PROGRAM SafetyCheck
VAR
	// slave robot information, including arm status and cartesian data
	m_slaveStatus AT %I* :ST_slaveStatus;
	
	// slave robot joint data
	m_slaveJointData AT %I* :ST_slaveJointData;
	
	// setup robot information
	m_setupStatus AT %I* :ST_SetupStatus;
	
	// setup robot joint data
	m_setupJointsData AT %I* :ST_SetupJointData;
	
	// master robot data, input from master controller box
	m_masterRobotData AT %I* : MSCommu_MasterStatus;
	
	// error check result
	m_safetyCheckData AT %Q* :ST_SafetyData;
	
	// Output cart status
	m_cartStatus AT%I* : ST_CartStatus;
	
	// cart joint data
	m_cartJointsData AT %I* :ST_CartJointData;
	
	//setup motor in_output to safety check
	m_setupMotorData AT %I* : ST_SetupMotorData;
	
	//slave motor in_output to safety check
	m_slaveMotorData AT %I* : ST_SlaveMotorData;
	
	//emergency stop and stop botton
	m_stopButton AT %I*: BOOL;
	m_emergencyStopButton AT %I*: BOOL;
	
	//warning tone
	m_warningTone AT %Q*:ARRAY [1..4] OF BOOL;
	
	//joystick Signal safety check
	m_joystickSignalIOSafetyCheck AT %I* : ARRAY [1..4] OF UDINT;
	
	//cart six-forceSensor
	m_sixForceSensor AT %I* : ARRAY [1..3] OF UDINT;
	
	//brake distance check outpurt
	m_brakeDistanceCheck AT %Q* : BOOL;
	
	i , j: INT;
	m_systemInitFlag:bool;
	m_SafetyCheck : Fb_SafetyCheck;
	m_clearFault : BOOL;
	m_checkVariable : ARRAY[1..g_maxNum] OF checkInputVariable;
	m_EtherCATCheck :ARRAY [1..g_maxNum,1..g_maxArmJoint] OF Fb_EtherCATCheck;
	m_EtherCATClearCRC :ARRAY [1..g_sArmNum] OF Fb_EtherCATCheck;
	m_RS232EtherCATState : ST_EtherCATState;
	
	//error robot data record
	m_dataRecord : Fb_dataRecord;
	
	// original position of remote center point when fisrt enter hold state
	m_dsrRcpPos :ARRAY[1..g_sArmNum] OF Vec3d;
	m_rcpPosErrCounts :ARRAY[1..g_sArmNum] OF INT := [4(0)];
	m_rcpPosErr :ARRAY[1..g_sArmNum] OF Vec3d;		// rcp position error
	m_motorEncoderSaltaValue : ARRAY [1..g_maxArmNum] OF vec13di;  
	
	m_armsRS:ARRAY [1..g_maxArmNum,1..50] OF RS;//复位优先双稳态器
	m_cartRS:ARRAY [1..50] OF RS;//复位优先双稳态器
	m_resetTon :ARRAY [1..g_maxArmNum,1..2] OF FB_TON;
	m_scopeArmNoReady : BOOL;
	m_joysticksTrigger : BOOL;
	// wait time before robot init  for ethercat to be statble 
	m_safetyCheckInitWaitTime : Vec5d;
	m_safetyCheckDriveOPWaitTime : LREAL:=0;
	m_safetyCheckReadFileWaitTime : LREAL:=0;
	
	m_EtherCATAllOP : BOOL:=FALSE;
	m_armEtherCATInOP : vec4b;
	m_moduleEtherCATInOPState : Vec5b;
	m_dumpEnergy : UDINT;
	
	m_mStopButton : FB_MasterStopButtonDetect;
	m_sStopButton : FB_MasterStopButtonDetect;
	
	//recipe read-write commands
	RecipeManCommands:   RecipeManCommands;
	m_bReadRecipeStep:   INT := 1;
	m_bWriteRecipeStep:   INT := 1;
	m_bReadRecipe:  BOOL := TRUE;
	m_bReadRecipeRecord:  BOOL := TRUE;
	
	m_bReadRecipeScope: BOOL := TRUE;
	
	m_bWriteRecipe: BOOL := FALSE;
	m_bWriteRecipeR: ARRAY [1..10] OF R_TRIG;
	m_ReturnDwordWrite : DWORD;
	m_loadConfigFileOK :BOOL :=FALSE;
	m_returnDwordRead:DWORD;
	m_returnDwordReadCart:DWORD;
	m_returnDwordReadMotorPara:DWORD;
	m_returnDwordReadReParam:DWORD;
	
	m_returnDwordReadScope:DWORD;
	
	m_caliFileWriteTon :ARRAY [1..g_sArmNum] OF TON ;
	m_linkPosWriteCaliData:ARRAY [1..4] OF ARRAY [1..8] OF TON ;
	m_powerBoxWriteCaliData:ARRAY [1..4] OF TON ;
	m_caliFileWriteTonOfCart :TON ;
	m_linkPosWriteCaliDataOfCart:ARRAY [1..8] OF TON ;

	
	//workHeart
	m_workHeartTon0 : TON;
	m_workHeartTon1 : TON;
	
	// flag if master are connected
	m_masterOnLine :BOOL :=FALSE;
	m_masterOnLineCheck :FB_masterConnectionCheck;
	
	//robot system operates sound 
	m_systemVoiceR:ARRAY [1..g_sArmNum,1..10] OF R_TRIG;
	m_systemVoiceF:ARRAY [1..g_sArmNum,1..10] OF F_TRIG;
	m_systemVoiceRS:ARRAY [1..g_sArmNum,1..10] OF RS;
	m_systemVoiceTon:ARRAY [1..g_sArmNum,1..10] OF FB_TON;
	m_checkArmKeepTriggerTon :ARRAY [1..g_sArmNum] OF FB_TON;
	m_trocarOnDetectTon:ARRAY [1..g_sArmNum] OF FB_TON;
	m_armStateLast:ARRAY[1..g_sArmNum] OF E_SlaveArmState;
	m_systemVoiceTriggerTime :TIME:=T#100MS;
	m_armKeepTriggerState :Vec4b;
	
	//read Net ID and Net port
	m_deviceNetIdReadOK : BOOL;
	m_bReadNetIdStep : INT := 1;
	m_bReadNetIdNum : INT := 1;
	m_bReadJntPortNum : INT := 1;
	m_getDeviceId :ARRAY [1..6] OF IOF_GetDeviceIDByName;
	m_getNetId :ARRAY [1..6] OF IOF_GetDeviceNetId;
	m_getBoxAddr:ARRAY [1..5,1..13] OF IOF_GetBoxAddrByName;
	m_readNetID: ARRAY[1..6] OF T_AmsNetId;
	m_readDeviceID : ARRAY [1..6]  OF UDINT;
	m_readJointNetPort:ARRAY[1..13] OF UINT;
END_VAR

// Faulty sound effect
m_warningTone := warningTone();
communicationCheck();
// reset data
m_deviceNetIdReadOK:=readDeviceNetId();
m_loadConfigFileOK:=loadConfigFile();
IF NOT(m_loadConfigFileOK) OR NOT m_deviceNetIdReadOK THEN
	m_safetyCheckReadFileWaitTime := m_safetyCheckReadFileWaitTime + g_safetyCheckCycleTime;
	IF m_safetyCheckReadFileWaitTime > g_robotSafetyReadFileWaitTime THEN
		GVL_interactUI.g_errIdType3:=checkFileAndNetId(m_loadConfigFileOK , m_deviceNetIdReadOK );
	END_IF
	RETURN;
END_IF
GVL_interactUI.g_systemVoice := systemVoice();

IF FALSE = m_systemInitFlag  THEN
	m_systemInitFlag := systemParaInit();
	RETURN;
END_IF

armSafetyCheckInputCast();

armSafetyCheckAllowed();

robotPromptMassageCast();

//robot record information
m_dataRecord.run(m_checkVariable , m_cartStatus , m_cartJointsData , m_setupStatus , m_slaveStatus , m_setupJointsData , m_slaveJointData );

//check EtherCAT status of arm and cart , if All EtherCAT is OP then start system safty check
IF FALSE = m_EtherCATAllOP THEN
	m_EtherCATAllOP := checkOPState();
END_IF

FOR i:=1  TO g_maxNum DO
	IF  NOT m_moduleEtherCATInOPState[i] AND NOT m_EtherCATAllOP THEN
		CONTINUE;
	END_IF
	
	// wait communication to be stable
	IF (m_safetyCheckInitWaitTime[i]<g_robotSafetyCheckWaitTime) THEN
		m_safetyCheckInitWaitTime[i] := m_safetyCheckInitWaitTime[i]+g_safetyCheckCycleTime;
	END_IF
	
	IF (m_safetyCheckInitWaitTime[i]>=g_robotSafetyCheckWaitTime) THEN
		m_SafetyCheck.systemSafetyCheck(i,m_checkVariable,m_cartJointsData,m_setupJointsData,m_slaveJointData);
	END_IF
END_FOR

//error flag to control
readErrFlag();

//Fault code for UI
m_SafetyCheck.errCodeUpdating();

//The fault code is sent to the UI
GVL_interactUI.g_errIdType3:=m_SafetyCheck.o_ErrCode[3];
GVL_interactUI.g_errIdType2:=m_SafetyCheck.o_ErrCode[2];
GVL_interactUI.g_errIdType1:=m_SafetyCheck.o_ErrCode[1];
GVL_interactUI.g_errIdType0:=m_SafetyCheck.o_ErrCode[0];
GVL_interactUI.g_popupErrorArm1 := m_SafetyCheck.m_armErrCodePopup[1];
GVL_interactUI.g_popupErrorArm2 := m_SafetyCheck.m_armErrCodePopup[2];
GVL_interactUI.g_popupErrorArm3 := m_SafetyCheck.m_armErrCodePopup[3];
GVL_interactUI.g_popupErrorArm4 := m_SafetyCheck.m_armErrCodePopup[4];

//clear fault
clearErrorFault();

METHOD armSafetyCheckAllowed : BOOL
VAR_INPUT
END_VAR
VAR
	i , j : INT; 
END_VAR
FOR i := 1 TO g_maxArmNum DO
	FOR j := 1 TO g_maxArmJoint DO
		IF j > 5 THEN
			//fault code 16#3003 
			m_SafetyCheck.checkPermit[i].m_linkEncErr[j] := m_checkVariable[i].m_slaveDriverInput[j-g_setupJntNum].m_statusWord<>0;
			//fault code 16#2002
			m_SafetyCheck.checkPermit[i].m_armJntFollowErr[j] := m_checkVariable[i].m_slaveDriverInput[j-g_setupJntNum].m_statusWord = DriverStatusWord_OP ;
			//fault code 16#200B
			m_SafetyCheck.checkPermit[i].m_jntCurrentCtrlErr[j] :=SlaveArmControl.m_slaveRobot.m_armCtrlCmds[i].m_jntEnableFlag[j-g_setupJntNum]  = DriverOPMode_Trq AND m_slaveMotorData.m_slaveMotorOutput[i,j-g_setupJntNum].m_opMode = DriverOPMode_Trq ;
		ELSE
			//fault code 16#3003 
			m_SafetyCheck.checkPermit[i].m_linkEncErr[j] := m_checkVariable[i].m_setupDriverInput[j].m_statusWord<>0;
			//fault code 16#2002
			m_SafetyCheck.checkPermit[i].m_armJntFollowErr[j] := m_checkVariable[i].m_setupDriverInput[j].m_statusWord = DriverStatusWord_OP AND j > 2;
			//fault code 16#200B
			m_SafetyCheck.checkPermit[i].m_jntCurrentCtrlErr[j] := SetupArmControl.m_setupRobot.m_armCtrlCmds[i].m_jntEnableFlag[j] = DriverOPMode_Trq AND m_setupMotorData.m_setupMotorOutput[i,j].m_opMode = DriverOPMode_Trq AND j > 2;
			
		END_IF
		//fault code 16#3002
		m_SafetyCheck.checkPermit[i].m_jntStatusErr[j] := TRUE;
		//fault code 16#3004
		m_SafetyCheck.checkPermit[i].m_driveErr[j] := TRUE;
		//fault code 16#3005
		m_SafetyCheck.checkPermit[i].m_armJntEncErr[j] := m_checkVariable[i].m_setupDriverInput[j].m_statusWord<>0;
		//fault code 16#3006
		m_SafetyCheck.checkPermit[i].m_outOfLimit[j] := m_checkVariable[i].m_setupDriverInput[j].m_statusWord<>0;
		//fault code 16#3008
		m_SafetyCheck.checkPermit[i].m_motPhieErr[j] := TRUE;
		//fault code 16#3009
		m_SafetyCheck.checkPermit[i].m_springBreakageCheck := TRUE;//m_checkVariable[i].m_setupDriverInput[j].m_statusWord<>0 ;
		//fault code 16#2003
		m_SafetyCheck.checkPermit[i].m_jntVelErr[j] := TRUE;
		//fault code 16#2004
		m_SafetyCheck.checkPermit[i].m_spacePoseErr := m_slaveStatus.m_armState[i] = SlaveArmState_MasterSlave;
		//fault code 16#2005
		m_SafetyCheck.checkPermit[i].m_jntCurrentErr[j] := TRUE;
		//fault code 16#2007
		m_SafetyCheck.checkPermit[i].m_fixedPointErr :=m_slaveStatus.m_armState[i] = SlaveArmState_MasterSlave;
		//fault code 16#2008
		m_SafetyCheck.checkPermit[i].m_cmdJntSaltation[j] := m_slaveStatus.m_armState[i] = SlaveArmState_MasterSlave;
		//fault code 16#200A
		m_SafetyCheck.checkPermit[i].m_simCmdSalta := m_slaveStatus.m_armState[i] = SlaveArmState_MasterSlave;
		//fault code 16#200F
		m_SafetyCheck.checkPermit[i].m_instruOpenAngle := FALSE;
		//fault code 16#2013
		m_SafetyCheck.checkPermit[i].m_jntLimitErr := m_slaveStatus.m_armState[i] = SlaveArmState_MasterSlave;
	END_FOR
END_FOR
END_METHOD

METHOD armSafetyCheckInputCast : BOOL
VAR_INPUT
END_VAR

VAR
	i , j: INT; 
END_VAR
FOR i := 1 TO g_maxArmNum DO
	//emergency stop 、stop button and ui stop 
	m_checkVariable[i].EmergencyStop := m_emergencyStopButton;
	m_checkVariable[i].PCStopButton := GVL_interactUI.g_stopButtonFormUI;
	m_checkVariable[i].SlaveStopButton := m_sStopButton.run(m_stopButton);
	m_checkVariable[i].MasterStopButton := m_mStopButton.run(m_masterRobotData.m_masterStopButton);
	
	IF NOT(m_slaveStatus.m_armState[i] = SlaveArmState_MasterSlave OR m_slaveStatus.m_armState[i] = SlaveArmState_EndoScope) THEN
		m_dsrRcpPos[i] := m_setupStatus.m_rcPos[i];
	END_IF
	m_checkVariable[i].m_rcpCheck := m_SafetyCheck.rcpErrCheck(m_dsrRcpPos[i],  m_setupStatus.m_rcPos[i], m_rcpPosErrCounts[i] ,m_rcpPosErr[i]);
	m_checkVariable[i].m_spacePoseErr := m_SafetyCheck.rotErrCheck(m_slaveStatus.m_masterSlavePoseError[i]);
	m_checkVariable[i].m_cmdArmPos := m_slaveStatus.m_simDHJntPos[i];

	//slave robot input cast
	FOR j:=1 TO  g_sJntNum DO 		
		m_checkVariable[i].m_slaveDriverInput[j] := m_slaveMotorData.m_slaveMotorInput[i,j];
		m_checkVariable[i].m_slaveDriverOutput[j] := m_slaveMotorData.m_slaveMotorOutput[i,j];
		m_checkVariable[i].m_EtherCATState[j+g_setupJntNum] := m_EtherCATCheck[i,j+g_setupJntNum].EtherCATVerify(GVL_SystemParameters.g_slaveArmNetID[i],GVL_SystemParameters.g_slaveJointNetPort[i,j]);
		m_checkVariable[i].m_motorEncoderSaltaValue[j+g_setupJntNum] := m_slaveMotorData.m_motorEncSalta[i][j];
	END_FOR
	
	//setup robot input cast
	FOR j:=1 TO  g_setupJntNum DO 	
		m_checkVariable[i].m_setupDriverInput[j] := m_setupMotorData.m_setupMotorInput[i,j];
		m_checkVariable[i].m_setupDriverOutput[j] := m_setupMotorData.m_setupMotorOutput[i,j];
		m_checkVariable[i].m_EtherCATState[j] := m_EtherCATCheck[i,j].EtherCATVerify(GVL_SystemParameters.g_slaveArmNetID[i],GVL_SystemParameters.g_setupJointNetPort[i,j]);
		m_checkVariable[i].m_motorEncoderSaltaValue[j] := m_setupMotorData.m_motorEncSalta[i][j];
	END_FOR
END_FOR


//setup robot in-out variable cast
FOR j:=1 TO  g_cartJntNum DO
	m_checkVariable[5].EmergencyStop := m_emergencyStopButton;
	m_checkVariable[5].PCStopButton := GVL_interactUI.g_stopButtonFormUI;
	m_checkVariable[5].SlaveStopButton := m_sStopButton.run(m_stopButton);
	m_checkVariable[5].m_cartDriverInput[j] := CartControl.m_cartRobot.m_slaveCart.m_cartJoints[j].m_motorInputs;
	m_checkVariable[5].m_cartDriverOutput[j] := CartControl.m_cartRobot.m_slaveCart.m_cartJoints[j].m_motorOutputs;
	m_checkVariable[5].m_cartEtherCATState[j] := m_EtherCATCheck[5,j].EtherCATVerify(GVL_SystemParameters.g_slaveCartNetID,GVL_SystemParameters.g_cartJointNetPort[j]);
END_FOR

//RS232 communication state
m_RS232EtherCATState := m_EtherCATCheck[5,9].EtherCATVerify(GVL_SystemParameters.g_slaveCartNetID,GVL_SystemParameters.g_cartJointNetPort[5]+1);

//output to ui
Gvl_io.g_emergencyStopButton := m_emergencyStopButton;
Gvl_io.g_stopButton := m_stopButton;
END_METHOD

METHOD checkEtherCATAll : BOOL
VAR_IN_OUT CONSTANT
	i_EtherCATState: ARRAY [1..g_maxNum] OF checkInputVariable;
END_VAR
VAR_OUTPUT
	o_EtherCATInOP : BOOL;
	o_armEtherCATInOP : vec4b;
	o_cartEtherCATAllOP : BOOL;
END_VAR

VAR
	i , j :INT;
END_VAR
FOR i := 1 TO g_sArmNum DO
	FOR j := 1 TO g_maxArmJoint DO
		//m_EtherCATCheck[i,j].setSlaveStatus(GVL_SlaveJointEncoderCaliData.g_slaveArmNetID[i],g_JointNetPort[j]);
	END_FOR
END_FOR

o_EtherCATInOP := TRUE;
FOR i := 1 TO g_sArmNum DO
	o_armEtherCATInOP[i] := TRUE;
	FOR j := 1 TO g_maxArmJoint DO
		IF FALSE = i_EtherCATState[i].m_EtherCATState[j].EtherCATState AND i <> GVL_interactUI.g_armIsDisable THEN
			o_armEtherCATInOP[i] := FALSE;
			o_EtherCATInOP := FALSE;
			EXIT;
		END_IF
	END_FOR
	IF NOT o_armEtherCATInOP[i] OR NOT o_EtherCATInOP THEN
		EXIT;
	END_IF
END_FOR

FOR j := 1 TO g_maxCartJoint DO
	//m_EtherCATCheck[5,j].setSlaveStatus(GVL_CartJointEncoderCaliData.g_slaveCartNetID,GVL_CartJointEncoderCaliData.g_slaveCartJointNetPort[j]);
END_FOR

o_cartEtherCATAllOP := TRUE;
FOR j := 1 TO g_maxCartJoint DO
	IF FALSE = i_EtherCATState[5].m_cartEtherCATState[j].EtherCATState THEN
		o_cartEtherCATAllOP := FALSE;
		EXIT;
	END_IF
END_FOR
END_METHOD

METHOD checkFileAndNetId : UDINT
VAR_IN_OUT CONSTANT
	i_readConfigFileStatus :BOOL;
	i_readDeviceNetIdStatus :BOOL;
END_VAR

IF NOT i_readConfigFileStatus OR NOT i_readDeviceNetIdStatus THEN
	checkFileAndNetId:=SHL(16#0C,24)+SHL(0,16)+16#300A;
END_IF
END_METHOD

METHOD checkOPState : BOOL
VAR_INPUT
END_VAR
IF (NOT m_safetyCheckData.m_armEtherCATAllOP OR NOT m_safetyCheckData.m_cartEtherCATAllOP) THEN
	m_safetyCheckDriveOPWaitTime := m_safetyCheckDriveOPWaitTime+g_safetyCheckCycleTime;
	IF m_safetyCheckDriveOPWaitTime > g_robotSafetyDriveOPWaitTime THEN
		 m_SafetyCheck.checkOPStatus(m_moduleEtherCATInOPState);
	END_IF
	RETURN;
END_IF
checkOPState := TRUE;
m_SafetyCheck.resetOPErrCode();
END_METHOD

METHOD clearErrorFault : BOOL
VAR_INPUT
END_VAR
VAR_STAT
	clearFaultTime : FB_TON;
END_VAR
// clear CRC lost frame
m_clearFault := GVL_interactUI.g_uiFaultReset=1 OR m_masterRobotData.m_uiResetFault = 1;
clearFaultTime(IN:= m_clearFault, PT:= T#2MS, Q=> , ET=> );
FOR i:=1 TO g_sArmNum DO 
	m_EtherCATClearCRC[i].clearCRCError(GVL_SystemParameters.g_slaveArmNetID[i],clearFault);
END_FOR
//clear fault
IF m_clearFault THEN
	m_SafetyCheck.errFlagReset();
	IF clearFaultTime.Q THEN
		GVL_interactUI.g_uiFaultReset := 0;
	END_IF
END_IF
END_METHOD

PROPERTY clearFault : BOOL;
GET
clearFault := m_clearFault;
END_GET
END_PROPERTY

METHOD communicationCheck : BOOL
VAR_INPUT
END_VAR
VAR
	i : INT;
END_VAR
checkEtherCATAll(m_checkVariable , o_EtherCATInOP=>m_safetyCheckData.m_armEtherCATAllOP,o_armEtherCATInOP=> m_armEtherCATInOP, o_cartEtherCATAllOP=> m_safetyCheckData.m_cartEtherCATAllOP );
FOR i := 1 TO g_sArmNum DO
	m_moduleEtherCATInOPState[i] := m_armEtherCATInOP[i];
END_FOR
m_moduleEtherCATInOPState[5] := m_safetyCheckData.m_cartEtherCATAllOP;

m_brakeDistanceCheck :=NOT UINT_TO_BOOL( GVL_interactUI.g_stopButtonFormUI);

//work heart
m_workHeartTon0(IN:= GVL_interactUI.g_heartBeat = 1, PT:= T#1S, Q=> , ET=> );
m_workHeartTon1(IN:= GVL_interactUI.g_heartBeat = 0, PT:= T#1S, Q=> , ET=> );
IF m_workHeartTon0.Q THEN
	GVL_interactUI.g_heartBeat :=0 ;
ELSIF m_workHeartTon1.Q THEN
	GVL_interactUI.g_heartBeat  :=1 ;
END_IF

//master online
m_masterOnLine := m_masterOnLineCheck.check(m_masterRobotData.m_heartBeat );

GVL_interactUI.g_slaveRunAlone := NOT m_masterOnLine;
END_METHOD

METHOD jointEncoderCaliCast : BOOL
VAR_INPUT
	armIdx : INT;
END_VAR
VAR 
	i : INT;
END_VAR

FOR i := 1 TO 8 DO
	m_linkPosWriteCaliData[armIdx][i](IN:= GVL_armCali.g_linkPosWriteCaliData[armIdx][i], PT:= T#3S, Q=> GVL_armCali.g_linkPosWriteCaliDataTrigger[armIdx][i], ET=> );
	IF GVL_armCali.g_linkPosWriteCaliDataTrigger[armIdx][i] THEN
		IF i<=5 THEN
			GVL_SetupJointEncoderCaliData.g_minLinkEncoder[armIdx,i] := GVL_armCali.g_linkLimitFristPos[armIdx][i];
			GVL_SetupJointEncoderCaliData.g_maxLinkEncoder[armIdx,i] := GVL_armCali.g_linkLimitSecondPos[armIdx][i];
			GVL_SetupJointEncoderCaliData.g_caliLinkEncoder[armIdx,i] := GVL_armCali.g_linkHomePos[armIdx][i];
			GVL_SetupJointEncoderCaliData.g_linkEncZeroCross[armIdx,i] := GVL_armCali.g_linkZeroCrossOrNot[armIdx][i];
		ELSE
			GVL_SlaveJointEncoderCaliData.g_minLinkEncoder[armIdx,i-5] := GVL_armCali.g_linkLimitFristPos[armIdx][i];
			GVL_SlaveJointEncoderCaliData.g_maxLinkEncoder[armIdx,i-5] := GVL_armCali.g_linkLimitSecondPos[armIdx][i];
			GVL_SlaveJointEncoderCaliData.g_caliLinkEncoder[armIdx,i-5] := GVL_armCali.g_linkHomePos[armIdx][i];
			GVL_SlaveJointEncoderCaliData.g_linkEncZeroCross[armIdx,i-5] := GVL_armCali.g_linkZeroCrossOrNot[armIdx][i];
		END_IF
	END_IF
END_FOR
FOR i := 1 TO 5 DO
	m_powerBoxWriteCaliData[armIdx](IN:= GVL_armCali.g_powerBoxPosWrite[armIdx], PT:= T#3S, Q=>GVL_armCali.g_powerBoxPosWriteTrigger[armIdx] , ET=> );
	IF GVL_armCali.g_powerBoxPosWriteTrigger[armIdx] THEN
		GVL_SlaveJointEncoderCaliData.g_caliLinkEncoder[armIdx,i+3] := GVL_armCali.g_powerBoxLinkHomePos[armIdx][i];
	END_IF
END_FOR

FOR i := 1 TO g_cartJntNum DO
	m_linkPosWriteCaliDataOfCart[i](IN:= GVL_armCali.g_linkPosWriteCaliDataOfCart[i], PT:= T#3S, Q=> GVL_armCali.g_linkPosWriteCaliDataTriggerOfCart[i], ET=> );
	IF GVL_armCali.g_linkPosWriteCaliDataTriggerOfCart[i] THEN
		GVL_CartJointEncoderCaliData.g_minLinkEncoder[i] := GVL_armCali.g_linkLimitFristPosOfCart[i];
		GVL_CartJointEncoderCaliData.g_maxLinkEncoder[i] := GVL_armCali.g_linkLimitSecondPosOfCart[i];
		GVL_CartJointEncoderCaliData.g_caliLinkEncoder[i] := GVL_armCali.g_linkHomePosOfCart[i];
		GVL_CartJointEncoderCaliData.g_linkEncZeroCross[i] := GVL_armCali.g_linkZeroCrossOrNotOfCart[i];
	END_IF
END_FOR
END_METHOD

METHOD joystickAdjust : BOOL
VAR_IN_OUT CONSTANT
	i_joystickValue : ARRAY [1..4] OF UDINT;
END_VAR

VAR
	i : INT;
END_VAR

FOR i := 1 TO 4 DO
	IF  (i_joystickValue[i]>1 AND i_joystickValue[i]<(512-50)) OR i_joystickValue[i] > (512+50) THEN
		joystickAdjust := TRUE;
		EXIT;
	END_IF
END_FOR
END_METHOD

METHOD loadConfigFile : BOOL
VAR
	i:INT;
	recordParam : BOOL;
	ReturnDwordWrite :DWORD;
END_VAR
//read recipe
IF (m_bReadRecipeStep<=12 AND m_bReadRecipeStep>0) THEN
	//The method loads a recipe from the specified recipe file.  It subsequently writes the recipe into the PLC variables.
    m_returnDwordRead:=RecipeManCommands.LoadAndWriteRecipe(RecipeDefinitionName:=GVL_SystemParameters.RecipeDefinitionName[m_bReadRecipeStep] , RecipeName:='RecipeRecord');
	IF m_returnDwordRead = ERR_OK THEN
		m_bReadRecipeStep:=m_bReadRecipeStep+1; 
	END_IF
END_IF 
loadConfigFile := m_bReadRecipeStep>12;


// read Recipe 
IF (m_bReadRecipe) THEN
	//The method loads a recipe from the specified recipe file.  It subsequently writes the recipe into the PLC variables.
     m_returnDwordReadCart:=RecipeManCommands.LoadAndWriteRecipe(RecipeDefinitionName:=GVL_SystemParameters.RecipeDefinitionNameCart, RecipeName:='RecipeRecord');	 
     m_returnDwordReadMotorPara:=RecipeManCommands.LoadAndWriteRecipe(RecipeDefinitionName:=GVL_SystemParameters.RecipeDefinitionNameMotorPara, RecipeName:='RecipeRecord');	
	m_bReadRecipe:=FALSE; 
END_IF
loadConfigFile := loadConfigFile AND (m_returnDwordReadCart = ERR_OK) AND m_returnDwordReadMotorPara = ERR_OK;

//read endoscope parameters
IF m_bReadRecipeScope THEN
	m_returnDwordReadScope:=RecipeManCommands.LoadAndWriteRecipe(RecipeDefinitionName:=GVL_SystemParameters.RecipeDefinitionNameScope, RecipeName:='RecipeRecord');	 
	m_bReadRecipeScope := FALSE;
END_IF
loadConfigFile := loadConfigFile AND m_returnDwordReadScope = ERR_OK;

//read robot record parameters
IF m_bReadRecipeRecord THEN
	m_returnDwordReadReParam:=RecipeManCommands.LoadAndWriteRecipe(RecipeDefinitionName:=GVL_SystemParameters.RecipeDefinitionNameRecordParam, RecipeName:='RecipeRecord');	 
	m_bReadRecipeRecord := FALSE;
END_IF


//write recipe
FOR i := 1 TO g_sArmNum DO
	jointEncoderCaliCast(i);
	m_caliFileWriteTon[i](IN:=GVL_armCali.g_caliDataWrite[i], PT:= T#3S, Q=> GVL_armCali.g_caliDataWriteTrigger[i], ET=> );
	IF GVL_armCali.g_caliDataWriteTrigger[i] THEN
		//This method creates a new recipe in the specified recipe definition. It subsequently reads the current PLC values into the new recipe and saves it as a recipe file with a standard name.
	 	RecipeManCommands.CreateRecipe(RecipeDefinitionName:=GVL_SystemParameters.RecipeDefinitionName[i] , RecipeName:='RecipeRecord' );
	 	ReturnDwordWrite:=RecipeManCommands.ReadAndSaveRecipe(RecipeDefinitionName:=GVL_SystemParameters.RecipeDefinitionName[i] , RecipeName:='RecipeRecord' );
	END_IF
END_FOR

m_caliFileWriteTonOfCart(IN:= GVL_armCali.g_caliDataWriteOfCart, PT:= T#3S, Q=> GVL_armCali.g_caliDataWriteTriggerOfCart, ET=> );
IF GVL_armCali.g_caliDataWriteTriggerOfCart THEN
	//This method creates a new recipe in the specified recipe definition. It subsequently reads the current PLC values into the new recipe and saves it as a recipe file with a standard name.
	 RecipeManCommands.CreateRecipe(RecipeDefinitionName:=GVL_SystemParameters.RecipeDefinitionNameCart , RecipeName:='RecipeRecord' );
	 ReturnDwordWrite:=RecipeManCommands.ReadAndSaveRecipe(RecipeDefinitionName:=GVL_SystemParameters.RecipeDefinitionNameCart , RecipeName:='RecipeRecord' );
	 m_bWriteRecipe:=FALSE;
END_IF

//write robot record parameters
FOR i := 1 TO g_sArmNum DO
	m_bWriteRecipeR[i](CLK:= MEMCMP(ADR(m_setupMotorData.m_jnt3MoveDistanceRecord[i]),ADR(m_setupMotorData.m_jnt3MoveDistance[i]),SIZEOF(m_setupMotorData.m_jnt3MoveDistanceRecord[i])) = 0, Q=> );
END_FOR
m_bWriteRecipeR[5](CLK:= MEMCMP(ADR(m_cartStatus.m_cartDriveForceOffset),ADR(m_cartStatus.m_cartDriveForceRecord),SIZEOF(m_cartStatus.m_cartDriveForceRecord)) = 0, Q=> );

m_bWriteRecipe := FALSE;
FOR i := 1 TO 10 DO
	IF m_bWriteRecipeR[i].Q THEN
		m_bWriteRecipe := m_bWriteRecipeR[i].Q;
		EXIT;
	END_IF
END_FOR

IF m_bWriteRecipe THEN
	 RecipeManCommands.CreateRecipe(RecipeDefinitionName:=GVL_SystemParameters.RecipeDefinitionNameRecordParam , RecipeName:='RecipeRecord' );
	 m_ReturnDwordWrite:=RecipeManCommands.ReadAndSaveRecipe(RecipeDefinitionName:=GVL_SystemParameters.RecipeDefinitionNameRecordParam , RecipeName:='RecipeRecord' );
END_IF
END_METHOD

METHOD readDeviceNetId : BOOL
VAR_INPUT
END_VAR
//read device NetId
CASE m_bReadNetIdStep OF
	1 ://read the device ID using the device name
		m_getDeviceId[m_bReadNetIdNum](NETID:= , DEVICENAME:= GVL_SystemParameters.g_deviceName[m_bReadNetIdNum], START:= TRUE, TMOUT:= , BUSY=> , ERR=> , ERRID=> , DEVICEID=> m_readDeviceID[m_bReadNetIdNum]);
		IF m_readDeviceID[m_bReadNetIdNum] <> 0 THEN
			m_bReadNetIdNum := m_bReadNetIdNum + 1;
			IF m_bReadNetIdNum > 6 THEN
				m_bReadNetIdNum:=1;
				m_bReadNetIdStep := 2;
			END_IF
		END_IF
		
	2:
		m_getNetId[m_bReadNetIdNum](NETID:= , DEVICEID:= m_readDeviceID[m_bReadNetIdNum], START:= TRUE, TMOUT:= , BUSY=> , ERR=> , ERRID=> , DeviceNetId=> m_readNetID[m_bReadNetIdNum]);
		IF m_readNetID[m_bReadNetIdNum] <> '' THEN
			IF m_bReadNetIdNum <= 4 THEN
				GVL_SystemParameters.g_slaveArmNetID [m_bReadNetIdNum] := m_readNetID[m_bReadNetIdNum];
				IF GVL_SystemParameters.g_slaveArmNetID [m_bReadNetIdNum] <> '' THEN
					m_bReadNetIdNum := m_bReadNetIdNum + 1;
				END_IF
			ELSIF m_bReadNetIdNum = 5 THEN
				GVL_SystemParameters.g_slaveCartNetID := m_readNetID[m_bReadNetIdNum];	
				IF GVL_SystemParameters.g_slaveCartNetID<> '' THEN
					m_bReadNetIdNum := m_bReadNetIdNum + 1;
				END_IF
			ELSIF m_bReadNetIdNum = 6 THEN
				GVL_SystemParameters.g_slaveMSComNetID := m_readNetID[m_bReadNetIdNum];	
				IF GVL_SystemParameters.g_slaveMSComNetID<> '' THEN
					m_bReadNetIdNum := m_bReadNetIdNum + 1;
				END_IF
			END_IF
			
			IF m_bReadNetIdNum > 6 THEN
				m_bReadNetIdNum:=1;
				m_bReadJntPortNum := 1;
				m_bReadNetIdStep := 3;
			END_IF
		END_IF
		
	3:
		IF m_bReadNetIdNum <= 4 THEN
			m_getBoxAddr[m_bReadNetIdNum,m_bReadJntPortNum](NETID:= , DEVICEID:= m_readDeviceID[m_bReadNetIdNum], BOXNAME:=GVL_SystemParameters.g_armDeviceJntName[m_bReadJntPortNum] , START:= TRUE, TMOUT:= , BUSY=> , ERR=> , ERRID=> , BOXADDR=> m_readJointNetPort[m_bReadJntPortNum]);
			IF m_bReadJntPortNum <= 5 THEN
				GVL_SystemParameters.g_setupJointNetPort[m_bReadNetIdNum,m_bReadJntPortNum] := m_readJointNetPort[m_bReadJntPortNum];
				IF GVL_SystemParameters.g_setupJointNetPort[m_bReadNetIdNum,m_bReadJntPortNum] <> 0 THEN
					m_bReadJntPortNum := m_bReadJntPortNum +1;
				END_IF
			ELSE
				GVL_SystemParameters.g_slaveJointNetPort[m_bReadNetIdNum,m_bReadJntPortNum-5]:= m_readJointNetPort[m_bReadJntPortNum];
				IF GVL_SystemParameters.g_slaveJointNetPort[m_bReadNetIdNum,m_bReadJntPortNum-5] <> 0 THEN
					m_bReadJntPortNum := m_bReadJntPortNum +1;
				END_IF
			END_IF
			IF m_bReadJntPortNum > 13 THEN
				m_bReadJntPortNum := 1;
				m_bReadNetIdNum := m_bReadNetIdNum + 1;
			END_IF
		ELSIF m_bReadNetIdNum = 5 THEN
			m_getBoxAddr[m_bReadNetIdNum,m_bReadJntPortNum](NETID:= , DEVICEID:= m_readDeviceID[m_bReadNetIdNum], BOXNAME:=GVL_SystemParameters.g_cartDeviceJntName[m_bReadJntPortNum] , START:= TRUE, TMOUT:= , BUSY=> , ERR=> , ERRID=> , BOXADDR=> m_readJointNetPort[m_bReadJntPortNum]);
				GVL_SystemParameters.g_cartJointNetPort[m_bReadJntPortNum] := m_readJointNetPort[m_bReadJntPortNum];
				IF GVL_SystemParameters.g_cartJointNetPort[m_bReadJntPortNum] <> 0 THEN
					m_bReadJntPortNum := m_bReadJntPortNum +1;
				END_IF
				IF m_bReadJntPortNum > 8 THEN
					m_bReadJntPortNum := 1;
					m_bReadNetIdNum := m_bReadNetIdNum + 1;
				END_IF
		END_IF
       
		IF m_bReadNetIdNum > 5 THEN
			m_bReadNetIdNum:=1;
			m_bReadNetIdStep := -1;
		END_IF
	
	-1:
		readDeviceNetId := TRUE;
END_CASE
END_METHOD

METHOD readErrFlag : BOOL
VAR_INPUT
END_VAR
FOR i:=1  TO g_sArmNum DO
	m_safetyCheckData.m_slaveErrFlag[i] := m_SafetyCheck.m_armErrFlag[i,2] OR m_SafetyCheck.m_armErrFlag[i,3];
	m_safetyCheckData.m_setupErrFlag[i] := m_SafetyCheck.m_armErrFlag[i,2] OR m_SafetyCheck.m_armErrFlag[i,3];
END_FOR


GVL_interactUI.g_slaveRecoverErrFlag := BOOL_TO_INT(((m_SafetyCheck.m_armErrFlag[1,2] AND GVL_interactUI.g_armIsDisable<>1) OR (m_SafetyCheck.m_armErrFlag[2,2] AND GVL_interactUI.g_armIsDisable<>2)
												 OR (m_SafetyCheck.m_armErrFlag[3,2] AND GVL_interactUI.g_armIsDisable<>3) OR (m_SafetyCheck.m_armErrFlag[4,2] AND GVL_interactUI.g_armIsDisable<>4)
														OR m_SafetyCheck.m_armErrFlag[g_cartNum,2] OR m_SafetyCheck.m_jntErrFlag[g_cartNum,0,2]) AND GVL_interactUI.g_slaveRunAlone) ;

//cart error flag
m_safetyCheckData.m_cartErrFlag := m_SafetyCheck.m_armErrFlag[g_cartNum,2] OR m_SafetyCheck.m_armErrFlag[g_cartNum,3];
//cart stead foot error flag
m_safetyCheckData.m_cartSteadyFootErr := m_SafetyCheck.m_jntErrFlag[g_cartNum,1,2] OR m_SafetyCheck.m_jntErrFlag[g_cartNum,1,3] 
																	OR m_SafetyCheck.m_jntErrFlag[g_cartNum,2,2] OR m_SafetyCheck.m_jntErrFlag[g_cartNum,2,3] OR m_SafetyCheck.m_jntErrFlag[g_cartNum,0,3];
//cart wheel error flag
m_safetyCheckData.m_cartWheelErr := m_SafetyCheck.m_jntErrFlag[g_cartNum,3,2] OR m_SafetyCheck.m_jntErrFlag[g_cartNum,3,3]
																OR m_SafetyCheck.m_jntErrFlag[g_cartNum,4,2] OR m_SafetyCheck.m_jntErrFlag[g_cartNum,4,3] OR m_SafetyCheck.m_stopButtonTrigger OR m_SafetyCheck.m_jntErrFlag[g_cartNum,0,3];
//cart stand column error flag
m_safetyCheckData.m_cartStandColumnErr := m_SafetyCheck.m_jntErrFlag[g_cartNum,5,2] OR m_SafetyCheck.m_jntErrFlag[g_cartNum,5,3] OR m_SafetyCheck.m_stopButtonTrigger OR m_SafetyCheck.m_jntErrFlag[g_cartNum,0,3];
//cart adjust joint contains 6, 7, and 8 joints
m_safetyCheckData.m_cartAdjustErr := m_SafetyCheck.m_jntErrFlag[g_cartNum,6,2] OR m_SafetyCheck.m_jntErrFlag[g_cartNum,6,3] 
															OR m_SafetyCheck.m_jntErrFlag[g_cartNum,7,2] OR m_SafetyCheck.m_jntErrFlag[g_cartNum,7,3]
															OR m_SafetyCheck.m_jntErrFlag[g_cartNum,8,2] OR m_SafetyCheck.m_jntErrFlag[g_cartNum,8,3] OR m_SafetyCheck.m_stopButtonTrigger OR m_SafetyCheck.m_jntErrFlag[g_cartNum,0,3];
//cart overhang error flag
m_safetyCheckData.m_cartOverhangErr := m_SafetyCheck.m_jntErrFlag[g_cartNum,8,2] OR m_SafetyCheck.m_jntErrFlag[g_cartNum,8,3] OR m_SafetyCheck.m_stopButtonTrigger OR m_SafetyCheck.m_jntErrFlag[g_cartNum,0,3];
END_METHOD

METHOD robotPromptMassageCast : BOOL
VAR_IN_OUT CONSTANT
END_VAR

VAR
	i : UDINT;
	m_uiCtrlAdjustFlag : BOOL;
	m_uiCtrlJoystickEnable : BOOL;
	instrument: INT;
	robotSelfCheckPass : BOOL;
	teleSlaveArmIdx : ARRAY [1..2] OF INT;
	panelMountedFlag : Vec4b;
	scopeNoReady : BOOL;
END_VAR
FOR i := 1 TO 4 DO
	//0*1021
	m_armsRS[i,1](SET:= m_slaveStatus.m_panelClampErrId[i]=1, 
							RESET1:= NOT m_slaveStatus.m_panelInstallStatus[i], 
							Q1=> m_checkVariable[i].m_promptStatus[1]);
	m_checkVariable[i].m_promptLocation[1] := i + 3;
							
	//0*1022		
	m_armsRS[i,2](SET:= m_slaveStatus.m_panelClampErrId[i]=2, 
							RESET1:= NOT m_slaveStatus.m_panelInstallStatus[i], 
							Q1=> m_checkVariable[i].m_promptStatus[2]);
	m_checkVariable[i].m_promptLocation[2] := i + 3;
	
	//0*1023				
	m_armsRS[i,3](SET:= m_slaveStatus.m_instruReadErrId[i]=1 AND m_slaveStatus.m_selfCheckPass[i], 
							RESET1:= NOT m_armsRS[i,3].SET OR NOT m_slaveStatus.m_instruInstallStatus[i] , 
							Q1=> m_checkVariable[i].m_promptStatus[3]);
	m_checkVariable[i].m_promptLocation[3] := i + 3;
						
	//0*1024	
	m_armsRS[i,4](SET:= m_slaveStatus.m_instruReadErrId[i]=2 AND m_slaveStatus.m_selfCheckPass[i],
							RESET1:=NOT m_armsRS[i,4].SET OR NOT m_slaveStatus.m_instruInstallStatus[i], 
							Q1=> m_checkVariable[i].m_promptStatus[4]);
	m_checkVariable[i].m_promptLocation[4] := i + 3;
	
	//0*1025
	m_armsRS[i,5](SET:= m_slaveStatus.m_instruClampErrId[i]=1 AND m_slaveStatus.m_selfCheckPass[i],
							RESET1:=NOT m_armsRS[i,5].SET OR NOT m_slaveStatus.m_instruInstallStatus[i], 
							Q1=> m_checkVariable[i].m_promptStatus[5]);
	m_checkVariable[i].m_promptLocation[5] := i + 3;
	
	 //0*1026
	m_armsRS[i,6](SET:= m_slaveStatus.m_instruClampErrId[i]=2 AND m_slaveStatus.m_selfCheckPass[i],
							RESET1:=NOT m_armsRS[i,6].SET OR NOT m_slaveStatus.m_instruInstallStatus[i], 
							Q1=> m_checkVariable[i].m_promptStatus[6]);
	m_checkVariable[i].m_promptLocation[6] := i + 3;
	
	//0*1027
	m_armsRS[i,7](SET:= m_slaveStatus.m_instruReadErrId[i]=3 AND m_slaveStatus.m_selfCheckPass[i],
							RESET1:=NOT m_armsRS[i,7].SET OR NOT m_slaveStatus.m_instruInstallStatus[i], 
							Q1=> m_checkVariable[i].m_promptStatus[7]);
	m_checkVariable[i].m_promptLocation[7] := i + 3;
	
	//0*1028	
	m_armsRS[i,8](SET:=NOT m_slaveStatus.m_selfCheckPass[i] AND m_slaveStatus.m_panelInstallStatus[i], 
							RESET1:= NOT m_armsRS[i,8].SET, 
							Q1=> m_checkVariable[i].m_promptStatus[8]);
	m_checkVariable[i].m_promptLocation[8] := i + 3;
				
	//0*1029
	m_armsRS[i,9](SET:= m_slaveStatus.m_instruReadErrId[i]=5 AND m_slaveStatus.m_selfCheckPass[i],
							RESET1:= NOT m_armsRS[i,9].SET OR NOT m_slaveStatus.m_instruInstallStatus[i], 
							Q1=> m_checkVariable[i].m_promptStatus[9]);
	m_checkVariable[i].m_promptLocation[9] := i + 3;
	
	 //0*102A
	m_armsRS[i,10](SET:= m_slaveStatus.m_instruReadErrId[i]=6 AND m_slaveStatus.m_selfCheckPass[i] AND NOT m_resetTon[i,1].Q,
							RESET1:= NOT m_armsRS[i,10].SET OR NOT m_slaveStatus.m_instruInstallStatus[i], 
							Q1=> m_checkVariable[i].m_promptStatus[10]);
	m_resetTon[i,1](IN:=m_slaveStatus.m_instruReadErrId[i]=6 AND m_slaveStatus.m_selfCheckPass[i] , PT:= T#5S, Q=> , ET=> );
	m_checkVariable[i].m_promptLocation[10] := i + 3;
	
	 //0*102B
	m_armsRS[i,11](SET:= m_slaveStatus.m_instruReadErrId[i]=4 AND m_slaveStatus.m_selfCheckPass[i] AND NOT m_resetTon[i,2].Q,
							RESET1:= NOT m_armsRS[i,11].SET, 
							Q1=> m_checkVariable[i].m_promptStatus[11]);
	m_resetTon[i,2](IN:=m_slaveStatus.m_instruReadErrId[i]=4 AND m_slaveStatus.m_selfCheckPass[i] , PT:= T#5S, Q=> , ET=> );
	m_checkVariable[i].m_promptLocation[11] := i + 3;	

	
	//0*102C
	m_armsRS[i,12](SET:= SlaveArmState_PanelReady= m_slaveStatus.m_armState[i] AND m_masterRobotData.m_tryMSControl[1] =1 AND m_slaveStatus.m_armState[i] <> SlaveArmState_Disable
							 AND m_slaveStatus.m_instruStauts[i].m_ready AND InstruType_endoscope <> m_slaveStatus.m_instruStauts[i].m_type AND m_setupStatus.m_armState[i] = SetupArmState_Hold , 
							RESET1:= NOT m_armsRS[i,12].SET, 
							Q1=> m_checkVariable[i].m_promptStatus[12]);
	m_checkVariable[i].m_promptLocation[12] := i + 3;

	
				
	//0*102D
	m_armsRS[i,13](SET:= norm(m_slaveStatus.m_masterSlavePoseError[i]) > g_smallNum AND m_slaveStatus.m_armState[i] = SlaveArmState_MasterSlave, 
							RESET1:= NOT m_armsRS[i,13].SET, 
							Q1=> m_checkVariable[i].m_promptStatus[13]);
	m_checkVariable[i].m_promptLocation[13] := i + 3;
	
	
	//0*102E
	m_armsRS[i,14](SET:= NOT SlaveArmControl.m_slaveRobot.m_panelMountedFlag[i] AND (m_masterRobotData.m_tryMSControl[1] =1 OR m_masterRobotData.m_tryMSControl[2] =1) AND m_slaveStatus.m_selfCheckPass[i],
							RESET1:= NOT m_armsRS[i,14].SET, 
							Q1=> m_checkVariable[i].m_promptStatus[14]);
	m_checkVariable[i].m_promptLocation[14] := i + 3;		
	
	//0*102F
	IF InstruType_endoscope = m_slaveStatus.m_instruStauts[i].m_type AND m_slaveStatus.m_endoscopeMounted THEN
		m_scopeArmNoReady :=  SlaveArmState_PanelReady= m_slaveStatus.m_armState[i] AND  m_slaveStatus.m_instruStauts[i].m_ready AND InstruType_endoscope = m_slaveStatus.m_instruStauts[i].m_type AND m_setupStatus.m_armState[i] = SetupArmState_Hold;
		m_armsRS[i,15](SET:= (NOT m_slaveStatus.m_endoscopeMounted OR m_scopeArmNoReady) AND (m_masterRobotData.m_tryMSControl[1] =1 OR m_masterRobotData.m_tryMSControl[2] =1), 
								RESET1:= NOT m_armsRS[i,15].SET, 
								Q1=> m_checkVariable[i].m_promptStatus[15]);
		m_checkVariable[i].m_promptLocation[15] := i + 3;	
	ELSE
		m_checkVariable[i].m_promptStatus[15] := FALSE;
		m_checkVariable[i].m_promptLocation[15] := i + 3;	
	END_IF
	
	//1037
	teleSlaveArmIdx := m_masterRobotData.m_teleSlaveArmIdx;
	IF InstruType_endoscope = m_slaveStatus.m_instruStauts[i].m_type AND m_slaveStatus.m_endoscopeMounted THEN
		scopeNoReady := NOT( SlaveArmState_ScopeReady= m_slaveStatus.m_armState[i] OR SlaveArmState_EndoScope= m_slaveStatus.m_armState[i]) OR NOT  m_slaveStatus.m_instruStauts[i].m_ready OR NOT InstruType_endoscope = m_slaveStatus.m_instruStauts[i].m_type ;
	END_IF
	FOR j:=1 TO g_mArmNum DO 
		IF i = teleSlaveArmIdx[j] THEN
			m_armsRS[i,23](SET:=m_slaveStatus.m_armState[i] = SlaveArmState_PanelReady AND m_masterRobotData.m_tryMSControl[j] =1 AND NOT m_slaveStatus.m_instruStauts[i].m_ready 
											 AND m_slaveStatus.m_endoscopeMounted AND NOT scopeNoReady, 
									RESET1:= NOT m_armsRS[i,23].SET, 
									Q1=> m_checkVariable[i].m_promptStatus[23]);
			m_checkVariable[i].m_promptLocation[23] := i + 3; EXIT;
		ELSE
			 m_checkVariable[i].m_promptStatus[23] := FALSE;
		END_IF
	END_FOR
	
	//1038
	//m_armsRS[i,24](SET:= SlaveArmControl.m_slaveRobot.panelMountedFlag[i] AND   (m_setupStatus.m_asepticMegnetCheck[i] AND 16#06) <> 16#06, 
	//						RESET1:= NOT m_armsRS[i,24].SET, 
	//						Q1=> m_checkVariable[i].m_promptStatus[24]);
	//m_checkVariable[i].m_promptLocation[24] := i + 3;
	
	//103C 内窥镜翻转中
	m_armsRS[i,28](SET:= SlaveArmState_ScopeToggle = m_slaveStatus.m_armState[i] AND SlaveArmControl.m_slaveRobot.m_scopeToggle[i].scopeIsTypeToggle = FALSE AND InstruType_endoscope = m_slaveStatus.m_instruStauts[i].m_type,
							RESET1:= NOT m_armsRS[i,28].SET, 
							Q1=> m_checkVariable[i].m_promptStatus[28]);
	m_checkVariable[i].m_promptLocation[28] := i + 3;
		
	//103D panel and instrument clamping at the same time
	m_armsRS[i,29](SET:=NOT SlaveArmControl.m_slaveRobot.m_panelMountedFlag[i] AND m_slaveStatus.m_selfCheckPass[i] AND m_slaveStatus.m_panelInstallStatus[i] AND m_slaveStatus.m_instruInstallStatus[i], 
							RESET1:= NOT m_armsRS[i,29].SET, 
							Q1=> m_checkVariable[i].m_promptStatus[29]);
	m_checkVariable[i].m_promptLocation[29] := i + 3;
	
	//1040 setup arm joint 3 spring check
	m_armsRS[i,32](SET:=m_setupMotorData.m_jnt3MoveDistanceRecord[i] > GVL_SafetyParameters.g_jnt3SpringLimit AND NOT m_slaveStatus.m_panelInstallStatus[i] , 
							RESET1:= NOT m_armsRS[i,32].SET, 
							Q1=> m_checkVariable[i].m_promptStatus[32]);
	m_checkVariable[i].m_promptLocation[32] := i + 3;
	
	//1041 mount instrument when slave arm is instrument retract state
	m_armsRS[i,33](SET:=SlaveArmState_InstruRetract = m_slaveStatus.m_armState[i] AND  SlaveArmControl.m_slaveRobot.m_SlaveArms[i].instruNear, 
							RESET1:= NOT m_armsRS[i,33].SET, 
							Q1=> m_checkVariable[i].m_promptStatus[33]);
	m_checkVariable[i].m_promptLocation[33] := i + 3;
END_FOR


//0*1030			
m_cartRS[16](SET:= NOT m_masterOnLine, 
						RESET1:= m_masterOnLine, 
						Q1=> m_checkVariable[g_cartNum].m_promptStatus[16]);
m_checkVariable[g_cartNum].m_promptLocation[16] := 16#0C;

//0*1031
IF NOT m_RS232EtherCATState.EtherCATState THEN
	m_dumpEnergy := 100;
ELSE
	m_dumpEnergy := GVL_interactUI.g_dumpEnergyUPS;
END_IF
m_cartRS[17](SET:=NOT SlaveArmControl.m_slaveInputDataPool.m_UIData.m_masterSlaveFlag AND GVL_interactUI.g_dumpEnergyUPS < 30 AND (m_masterRobotData.m_tryMSControl[1] =1 OR m_masterRobotData.m_tryMSControl[2] =1), 
						RESET1:=  SlaveArmControl.m_slaveInputDataPool.m_UIData.m_masterSlaveFlag OR  GVL_interactUI.g_dumpEnergyUPS >= 30 OR NOT (m_masterRobotData.m_tryMSControl[1] =1 OR m_masterRobotData.m_tryMSControl[2] =1), 
						Q1=> m_checkVariable[g_cartNum].m_promptStatus[17]);
m_checkVariable[g_cartNum].m_promptLocation[17] := g_cartNum + 3;

//0*1032	 没有卡接内窥镜时的检测	
FOR i := 1 TO g_sArmNum DO
	panelMountedFlag[i] := SlaveArmControl.m_slaveRobot.m_panelMountedFlag[i] OR i = GVL_interactUI.g_armIsDisable;
END_FOR
robotSelfCheckPass := panelMountedFlag[1] AND panelMountedFlag[2] AND panelMountedFlag[3] AND panelMountedFlag[4];
m_cartRS[18](SET:= robotSelfCheckPass AND  NOT m_slaveStatus.m_endoscopeMounted AND (m_masterRobotData.m_tryMSControl[1] =1 OR m_masterRobotData.m_tryMSControl[2] =1), 
						RESET1:= NOT m_cartRS[18].SET, 
						Q1=> m_checkVariable[g_cartNum].m_promptStatus[18]);
m_checkVariable[g_cartNum].m_promptLocation[18] := 16#0C;

//0*1033
m_cartRS[19](SET:= m_cartStatus.m_sdrivingLeverSensorManualFlag, 
						RESET1:=NOT m_cartStatus.m_sdrivingLeverSensorManualFlag, 
						Q1=> m_checkVariable[g_cartNum].m_promptStatus[19]);
m_checkVariable[g_cartNum].m_promptLocation[19] := g_cartNum + 3;

 //0*1034
m_uiCtrlJoystickEnable := m_cartStatus.m_uiControl.m_cameraJoystickEnable OR m_cartStatus.m_uiControl.m_joystickEnable OR m_cartStatus.m_uiControl.m_heightLimitAdjustEnable;
m_joysticksTrigger :=  joystickAdjust(m_joystickSignalIOSafetyCheck);
m_cartRS[20](SET:= m_cartStatus.m_trocarOnFlag=0 AND NOT m_uiCtrlJoystickEnable AND m_joysticksTrigger, 
						RESET1:= NOT m_cartRS[20].SET, 
						Q1=> m_checkVariable[g_cartNum].m_promptStatus[20]);
m_checkVariable[g_cartNum].m_promptLocation[20] := g_cartNum + 3;
					
//0*1035
m_uiCtrlAdjustFlag := m_cartStatus.m_uiControl.m_cameraJoystickEnable OR m_cartStatus.m_uiControl.m_dockingEnable OR m_cartStatus.m_uiControl.m_drapingEnable
							OR m_cartStatus.m_uiControl.m_joystickEnable OR m_cartStatus.m_uiControl.m_packageEnable OR CartControl.m_cartRobot.m_carHandChassisDriveUnlock[1] OR CartControl.m_cartRobot.m_carHandChassisDriveUnlock[2];
m_cartRS[21](SET:= m_cartStatus.m_trocarOnFlag>0 AND (m_uiCtrlAdjustFlag OR m_joysticksTrigger), 
						RESET1:= m_cartStatus.m_trocarOnFlag=0 OR (NOT m_uiCtrlAdjustFlag AND NOT m_joysticksTrigger), 
						Q1=> m_checkVariable[g_cartNum].m_promptStatus[21]);
m_checkVariable[g_cartNum].m_promptLocation[21] := g_cartNum + 3;

//0*1036
m_cartRS[22](SET:=  (m_cartStatus.m_jntPosReachLimit[5] OR m_cartStatus.m_jntPosReachLimit[6] OR m_cartStatus.m_jntPosReachLimit[7] OR m_cartStatus.m_jntPosReachLimit[8]), 
						RESET1:= NOT m_cartRS[22].SET, 
						Q1=> m_checkVariable[g_cartNum].m_promptStatus[22]);
m_checkVariable[g_cartNum].m_promptLocation[22] := g_cartNum + 3;

//0*1039
//m_cartRS[22](SET:=  (m_cartStatus.m_jntPosReachLimit[5] OR m_cartStatus.m_jntPosReachLimit[6] OR m_cartStatus.m_jntPosReachLimit[7] OR m_cartStatus.m_jntPosReachLimit[8]), 
//						RESET1:= NOT m_cartRS[22].SET, 
//						Q1=> m_checkVariable[g_cartNum].m_promptStatus[22]);
//m_checkVariable[g_cartNum].m_promptLocation[22] := g_cartNum + 3;
					
//0*103A
m_cartRS[26](SET:= m_joystickSignalIOSafetyCheck[1] = 0 OR m_joystickSignalIOSafetyCheck[2] = 0 OR m_joystickSignalIOSafetyCheck[3] = 0 OR m_joystickSignalIOSafetyCheck[4] = 0, 
						RESET1:= NOT m_cartRS[26].SET, 
						Q1=> m_checkVariable[g_cartNum].m_promptStatus[26]);
m_checkVariable[g_cartNum].m_promptLocation[26] := g_cartNum + 3;

//0*103B
m_cartRS[27](SET:= (m_sixForceSensor[1] = 0 OR m_sixForceSensor[2] = 0 OR m_sixForceSensor[3] = 0 ) AND m_cartStatus.m_CartState = CartJointState_Movement, 
						RESET1:= NOT m_cartRS[27].SET, 
						Q1=> m_checkVariable[g_cartNum].m_promptStatus[27]);
m_checkVariable[g_cartNum].m_promptLocation[27] := g_cartNum + 3;

//0*103E
m_cartRS[30](SET:= NOT CartControl.m_cartRobot.m_slaveCart.driveForceCaliState, 
						RESET1:= NOT m_cartRS[30].SET, 
						Q1=> m_checkVariable[g_cartNum].m_promptStatus[30]);
m_checkVariable[g_cartNum].m_promptLocation[30] := g_cartNum + 3;

//0*103F
m_cartRS[31](SET:= m_cartStatus.m_supportLegErrID[1]=2 OR m_cartStatus.m_supportLegErrID[2]=2, 
						RESET1:= NOT m_cartRS[31].SET, 
						Q1=> m_checkVariable[g_cartNum].m_promptStatus[31]);
m_checkVariable[g_cartNum].m_promptLocation[31] := g_cartNum + 3;
END_METHOD

PROPERTY safetyCheckData : REFERENCE TO ST_SafetyData
GET
safetyCheckData ref=m_safetyCheckData;
END_GET
END_PROPERTY

PROPERTY stopErrFlag : BOOL;
GET
stopErrFlag := m_SafetyCheck.m_stopButtonTrigger;
END_GET
END_PROPERTY

METHOD systemParaInit : BOOL
VAR_INPUT
END_VAR
VAR
	i, j : INT;
	cartJointPara : ST_CartJointParametersData;
	slaveArmJointPara :ST_slaveArmJointParametersData;
END_VAR
//reset error flag
FOR i:=1  TO g_sArmNum DO 
	m_safetyCheckData.m_slaveErrFlag[i]:=FALSE;
	m_safetyCheckData.m_setupErrFlag[i]:=FALSE;
END_FOR
m_safetyCheckData.m_cartErrFlag:=FALSE;
//**********************slave arm joint parameters ***************************//
IF g_slaveArmJointParametersVer = 'Ver2'  THEN
	slaveArmJointPara := g_systemArmJointPara.m_slaveArmJointParaVer2;
ELSE
	slaveArmJointPara := g_systemArmJointPara.m_slaveArmJointParaVer1;
END_IF

//slave arm joint parameters data initialize
GVL_SlaveMotorParameters.g_incEncoderRes := slaveArmJointPara.m_incEncoderRes;
GVL_SlaveMotorParameters.g_absEncoderRes := slaveArmJointPara.m_absEncoderRes;
GVL_SlaveMotorParameters.g_motorReduction := slaveArmJointPara.m_motorReduction;
GVL_SlaveMotorParameters.g_absEncoderReduction := slaveArmJointPara.m_absEncoderReduction;
GVL_SlaveMotorParameters.g_motorTrqConst := slaveArmJointPara.m_motorTrqConst;
GVL_SlaveMotorParameters.g_motorMaxCurrent := slaveArmJointPara.m_motorMaxCurrent;
GVL_SlaveMotorParameters.g_motorDir := slaveArmJointPara.m_motorDir;
GVL_SlaveMotorParameters.g_asbEncoderDir := slaveArmJointPara.m_asbEncoderDir;
GVL_SlaveMotorParameters.g_minJntPos := slaveArmJointPara.m_minJntPos;
GVL_SlaveMotorParameters.g_maxJntPos := slaveArmJointPara.m_maxJntPos;
GVL_SlaveMotorParameters.g_minDHJntPos := slaveArmJointPara.m_minDHJntPos;
GVL_SlaveMotorParameters.g_maxDHJntPos := slaveArmJointPara.m_maxDHJntPos;
GVL_SlaveMotorParameters.g_maxJntVel := slaveArmJointPara.m_maxJntVel;
GVL_SlaveMotorParameters.g_linkEncCaliJntPos := slaveArmJointPara.m_linkEncCaliJntPos;
GVL_SlaveMotorParameters.g_minInstruRCDis := slaveArmJointPara.m_minInstruRCDis;
GVL_SlaveMotorParameters.g_minScopeRCDis := slaveArmJointPara.m_minScopeRCDis;



//**********************Cart joint parameters ***************************//
//cart joint parameters version selection
IF g_cartJointParametersVer = 'Ver2'  THEN
	cartJointPara := g_systemArmJointPara.m_cartJointParaVer2;
ELSE
	cartJointPara := g_systemArmJointPara.m_cartJointParaVer1;
END_IF

//cart joint parameters data initialize
GVL_CartMotorParameters.g_incEncoderRes := cartJointPara.m_incEncoderRes;
GVL_CartMotorParameters.g_absEncoderRes := cartJointPara.m_absEncoderRes;
GVL_CartMotorParameters.g_motorReduction := cartJointPara.m_motorReduction;
GVL_CartMotorParameters.g_absEncoderReduction := cartJointPara.m_absEncoderReduction;
GVL_CartMotorParameters.g_motorTrqConst := cartJointPara.m_motorTrqConst;
GVL_CartMotorParameters.g_asbEncoderDir := cartJointPara.m_asbEncoderDir;
GVL_CartMotorParameters.g_motorTrqConst := cartJointPara.m_motorTrqConst;
GVL_CartMotorParameters.g_motorMaxCurrent := cartJointPara.m_motorMaxCurrent;
GVL_CartMotorParameters.g_motorDir := cartJointPara.m_motorDir;
GVL_CartMotorParameters.g_minJntPos := cartJointPara.m_minJntPos;
GVL_CartMotorParameters.g_maxJntPos := cartJointPara.m_maxJntPos;

systemParaInit := TRUE;
END_METHOD

METHOD systemVoice : INT
VAR_INPUT
END_VAR
VAR
	i : INT;
END_VAR
VAR_STAT
	panelInstalled : Vec4b;
	instruCtrlAdjust : Vec4b;
	instruCtrlAdjustFallEdge : Vec4b;
	manualCtrlAdjust : Vec4b;
	manualCtrlAdjustFallEdge : Vec4b;
	trocarInstalled : Vec4b;
	instruInstalled : Vec4b;
	instruInvasion : Vec4b;
END_VAR
FOR i := 1 TO g_sArmNum DO
	//panel installed succeed 
	m_systemVoiceR[i,1](CLK:=SlaveArmControl.m_slaveRobot.m_panelMountedFlag[i]  , Q=> );
	IF m_systemVoiceR[i,1].Q THEN
		panelInstalled[i]:=TRUE;
	END_IF
	m_systemVoiceTon[i,1](IN:= panelInstalled[i], PT:= m_systemVoiceTriggerTime, Q=> , ET=> );
	m_systemVoiceRS[i,1](SET:= panelInstalled[i], RESET1:= m_systemVoiceTon[i,1].Q , Q1=> );
	IF m_systemVoiceRS[i,1].Q1 THEN
		systemVoice := systemVoice_triger3;
		RETURN;
	ELSE
		panelInstalled[i]:=FALSE;
	END_IF

	//adjust button trigger and slave arm state at SlaveArmState_Adjust status
	m_systemVoiceR[i,2](CLK:= m_slaveStatus.m_armState[i] = SlaveArmState_Adjust, Q=> );
	IF m_systemVoiceR[i,2].Q THEN
		instruCtrlAdjust[i] := TRUE;
	END_IF
	m_systemVoiceTon[i,2](IN:= instruCtrlAdjust[i], PT:= m_systemVoiceTriggerTime, Q=> , ET=> );
	m_systemVoiceRS[i,2](SET:= instruCtrlAdjust[i], RESET1:= m_systemVoiceTon[i,2].Q , Q1=> );
	IF m_systemVoiceRS[i,2].Q1 THEN
		systemVoice := systemVoice_end4;
		RETURN;
	ELSE
		instruCtrlAdjust[i] := FALSE;
	END_IF
	
	//slave arm state exit SlaveArmState_Adjust status
	m_checkArmKeepTriggerTon[i](IN:=NOT SlaveArmControl.m_slaveRobot.m_slaveArms[i].adjustOn AND m_slaveStatus.m_armState[i] = SlaveArmState_Adjust, PT:= T#0.01S, Q=> , ET=> );
	IF m_checkArmKeepTriggerTon[i].Q THEN
		m_armKeepTriggerState[i]:=TRUE;
	END_IF
	m_systemVoiceF[i,3](CLK:=m_armKeepTriggerState[i] AND m_slaveStatus.m_armState[i] = SlaveArmState_Adjust, Q=> );
	IF m_systemVoiceF[i,3].Q THEN
		instruCtrlAdjustFallEdge[i] := TRUE;
	END_IF
	m_systemVoiceTon[i,3](IN:= instruCtrlAdjustFallEdge[i], PT:= m_systemVoiceTriggerTime, Q=> , ET=> );
	m_systemVoiceRS[i,3](SET:= instruCtrlAdjustFallEdge[i], RESET1:= m_systemVoiceTon[i,3].Q , Q1=> );
	IF m_systemVoiceRS[i,3].Q1 THEN
		systemVoice := systemVoice_end4;
		m_armKeepTriggerState[i]:=FALSE;
		RETURN;
	ELSE
		instruCtrlAdjustFallEdge[i] := FALSE;
	END_IF
	
	//adjust button trigger and setup arm state at SetupArmState_ManualAdjust status
	//m_systemVoiceR[i,4](CLK:=SetupArmControl.m_setupRobot.m_setupArms[i].manualAdjustOn AND m_setupStatus.m_armState[i] = SetupArmState_ManualAdjust, Q=> );
	//IF m_systemVoiceR[i,4].Q THEN
	//	manualCtrlAdjust[i] := TRUE;
	//END_IF
	//m_systemVoiceTon[i,4](IN:= manualCtrlAdjust[i], PT:= m_systemVoiceTriggerTime, Q=> , ET=> );
	//m_systemVoiceRS[i,4](SET:= manualCtrlAdjust[i], RESET1:= m_systemVoiceTon[i,4].Q , Q1=> );
	//IF m_systemVoiceRS[i,4].Q1 THEN
	//	systemVoice := systemVoice_end4;
	//	RETURN;
	//ELSE
	//	manualCtrlAdjust[i] := FALSE;
	//END_IF
	
	//slave arm state exit SetupArmState_ManualAdjust status
	//m_systemVoiceF[i,5](CLK:= SetupArmControl.m_setupRobot.m_setupArms[i].manualAdjustOn AND m_setupStatus.m_armState[i] = SetupArmState_ManualAdjust, Q=> );
	//IF m_systemVoiceF[i,5].Q THEN
	//	manualCtrlAdjustFallEdge[i] := TRUE;
	//END_IF
	//m_systemVoiceTon[i,5](IN:= manualCtrlAdjustFallEdge[i], PT:= m_systemVoiceTriggerTime, Q=> , ET=> );
	//m_systemVoiceRS[i,5](SET:= manualCtrlAdjustFallEdge[i], RESET1:= m_systemVoiceTon[i,5].Q , Q1=> );
	//IF m_systemVoiceRS[i,5].Q1 THEN
	//	systemVoice := systemVoice_end4;
	//	RETURN;
	//ELSE
	//	manualCtrlAdjustFallEdge[i] := FALSE;
	//END_IF
	
	//trocar installed
	m_trocarOnDetectTon[i](IN:= m_slaveStatus.m_trocarOnFlag[i], PT:= T#1S, Q=> trocarInstalled[i], ET=> );
	m_systemVoiceTon[i,6](IN:= trocarInstalled[i], PT:= m_systemVoiceTriggerTime, Q=> , ET=> );
	m_systemVoiceRS[i,6](SET:= trocarInstalled[i], RESET1:= m_systemVoiceTon[i,6].Q OR NOT trocarInstalled[i], Q1=> );
	IF m_systemVoiceRS[i,6].Q1 THEN
		systemVoice := systemVoice_triger3;
		RETURN;
	END_IF
	
	//instrument or endoscope installed
	m_systemVoiceR[i,7](CLK:=SlaveArmControl.m_slaveRobot.m_instrumentMountedFlag[i]  , Q=> );
	IF m_systemVoiceR[i,7].Q THEN
		instruInstalled[i]:=TRUE;
	END_IF
	m_systemVoiceTon[i,7](IN:= instruInstalled[i], PT:= m_systemVoiceTriggerTime, Q=> , ET=> );
	m_systemVoiceRS[i,7](SET:= instruInstalled[i], RESET1:= m_systemVoiceTon[i,7].Q , Q1=> );
	IF m_systemVoiceRS[i,7].Q1 THEN
		systemVoice := systemVoice_triger3;
		RETURN;
	ELSE
		instruInstalled[i]:=FALSE;
	END_IF
	
	//slave arm state exit SlaveArmState_InstruInvasion status
	m_systemVoiceR[i,8](CLK:= m_armStateLast[i] =SlaveArmState_InstruInvasion AND (m_slaveStatus.m_armState[i] = SlaveArmState_PanelReady OR m_slaveStatus.m_armState[i] = SlaveArmState_InstruReady), Q=> );
	IF m_systemVoiceR[i,8].Q THEN
		instruInvasion[i] := TRUE;
	END_IF
	m_armStateLast[i] := m_slaveStatus.m_armState[i];
	m_systemVoiceTon[i,8](IN:= instruInvasion[i], PT:= m_systemVoiceTriggerTime, Q=> , ET=> );
	m_systemVoiceRS[i,8](SET:= instruInvasion[i], RESET1:= m_systemVoiceTon[i,8].Q , Q1=> );
	IF m_systemVoiceRS[i,8].Q1 THEN
		systemVoice := systemVoice_triger3;
		RETURN;
	ELSE
		instruInvasion[i] := FALSE;
	END_IF
END_FOR
END_METHOD

METHOD warningTone : vec4b
VAR_INPUT
END_VAR
VAR
	i : INT;
	armStateIsPackage : BOOL;
END_VAR
FOR i := 1 TO g_sArmNum DO
	IF m_slaveStatus.m_armState[i] = SlaveArmState_Package OR (m_setupStatus.m_armState[i] = SetupArmState_AutoAdjust AND SetupArmControl.m_setupRobot.m_setupArms[i].jnt5AdjustDir <> 0) THEN
		armStateIsPackage := TRUE;
		EXIT;
	END_IF
END_FOR

IF (GVL_interactUI.g_curErrType=3) OR Gvl_io.g_openWarningTone[3] THEN
	warningTone[1] := TRUE;
	warningTone[2] := FALSE;
	warningTone[3] := FALSE;
ELSIF (GVL_interactUI.g_curErrType=2) OR Gvl_io.g_openWarningTone[2] THEN
	warningTone[1] := FALSE;
	warningTone[2] := TRUE;
	warningTone[3] := FALSE;
ELSIF (m_cartStatus.m_jntPosReachLimit[5] OR m_cartStatus.m_jntPosReachLimit[6] OR m_cartStatus.m_jntPosReachLimit[7] OR m_cartStatus.m_jntPosReachLimit[8]) THEN 
	warningTone[1] := FALSE;
	warningTone[2] := TRUE;
	warningTone[3] := TRUE;
ELSIF (m_cartStatus.m_CartState >= CartJointState_HangAdjust AND  m_cartStatus.m_CartState <= CartJointState_RotaOverhang) OR m_cartStatus.m_CartState = CartJointState_StandColuAdjust OR armStateIsPackage  OR Gvl_io.g_openWarningTone[4] THEN
	warningTone[1] := TRUE;
	warningTone[2] := FALSE;
	warningTone[3] := TRUE;
	
ELSIF (ABS(CartControl.m_cartRobot.m_slaveCart.m_columnJntVel) > g_smallNum AND NOT CartControl.m_cartRobot.m_slaveCart.m_columnAdjustEnable) OR Gvl_io.g_openWarningTone[5] THEN
	warningTone[1] := FALSE;
	warningTone[2] := FALSE;
	warningTone[3] := TRUE;

ELSIF (GVL_interactUI.g_curErrType=1) OR Gvl_io.g_openWarningTone[1] THEN
	warningTone[1] := TRUE;
	warningTone[2] := TRUE;
	warningTone[3] := FALSE;
ELSE
	warningTone[1] := FALSE;
	warningTone[2] := FALSE;
	warningTone[3] := FALSE;
END_IF
END_METHOD

END_PROGRAM

(* stored: Version 1.1.0.1, ProductVersion 3.1.4024.11
   POU SafetyCheck: Id {54e6e883-3f22-4a40-9066-2b433bf8009c}, SpecialFunc None
   Folder property: Id {5eb59b4d-8ad0-4d0f-a50e-7d8df12adfd3}
   Method armSafetyCheckAllowed: Id {c2ebef6f-e712-49e3-9955-377a0083e93a}
   Method armSafetyCheckInputCast: Id {598e934b-b439-4bef-985d-1ea697c2fcb0}
   Method checkEtherCATAll: Id {a164738b-81a3-4c66-88e6-d907208d76aa}
   Method checkFileAndNetId: Id {8c537d8f-f839-471c-bd2e-5b10d7fe3d04}
   Method checkOPState: Id {b7355243-ae6f-4b58-96ae-86072ab041c7}
   Method clearErrorFault: Id {4538f7d4-f9eb-4e43-b333-a31d3b56574d}
   Property clearFault: Id {62f202d3-4bb7-408a-b265-9c35a33c392a}
   Get Get: Id {d6f5c8ed-e672-4c40-9a2f-a6c375e1a742}
   Method communicationCheck: Id {50ac3c80-6bd7-4832-ad7c-bbfbaa36f395}
   Method jointEncoderCaliCast: Id {38e8df63-8a70-4816-82e7-e0e3cbf778d9}
   Method joystickAdjust: Id {38ce96d9-75fc-4e3b-9d39-89b30533a7ac}
   Method loadConfigFile: Id {a9343549-3fa6-461f-98d4-d8ffc4dbad86}
   Method readDeviceNetId: Id {0e6e0f21-760b-4ac7-b092-18d2817302c2}
   Method readErrFlag: Id {c6c3fbb5-bc5f-41ea-91b5-687651d637ca}
   Method robotPromptMassageCast: Id {4528e69f-5454-4a94-84aa-1a99d7ab54e4}
   Property safetyCheckData: Id {e78c5e7a-1511-4ab6-aa25-f80be9843ba9}
   Get Get: Id {9764d763-bd8c-45a4-8ee7-eb2346d1771d}
   Property stopErrFlag: Id {788bf35b-8072-4270-b764-825efb5a53e7}
   Get Get: Id {9923caa9-0191-4fd7-9dfb-98cb92ebe1ae}
   Method systemParaInit: Id {fe5c0617-d1df-4b96-8905-b301ef6249be}
   Method systemVoice: Id {1acc2045-db42-420c-8757-38d389cdc385}
   Method warningTone: Id {82112973-2b93-4990-831a-9a609be275a4} *)
